(* CODESYS project Kontrolki2.project

Project tree, tasks and I/O mapping:
  Device : CODESYS Control Win V3, 3S - Smart Software Solutions GmbH, order no. 305021, version 3.5.8.10
    application Application
      libraries: Standard, * (System)
      task MainTask (cyclic, interval t#20ms, priority 1) calls PLC_PRG
      task VISU_TASK (cyclic, interval 100 ms, priority 31) calls VisuElems.Visu_Prg
      program PLC_PRG [LD]
      visualisation Visualization
  libraries: VisuSymbols, 3.5.8.0 (System)
  text list GlobalTextList
*)

// Device/Application/PLC_PRG
PROGRAM PLC_PRG
VAR
	SET: BOOL;
	RESET: BOOL;
	//KONTROLKA 1 - CZERWONY
	K1: BOOL;
	//KONTROLKA 2 - ZIELONY
	K2: BOOL;
	//KONTROLKA 3 - NIEBIESKI
	K3: BOOL;
	//KONTROLKA 4 - ŻÓŁTY
	K4: BOOL;
	HOLD: BOOL;
	//SPRAWDZENIE CZY SIĘ ŚWIECI K1
	C1: BOOL;
	//SPRAWDZENIE CZY SIĘ ŚWIECI K2
	C2: BOOL;
	//SPRAWDZENIE CZY SIĘ ŚWIECI K3
	C3: BOOL;
	//SPRAWDZENIE CZY SIĘ ŚWIECI K4
	C4: BOOL;
	TON_K1: TON;
	TON_K2: TON;
	TON_K3: TON;
	CZAS: TIME;
	//SPRAWDZENIE CZY NACIŚNIĘTO RESET
	CHECK: BOOL;
END_VAR
VAR // added by the converter: edge detectors and wires of the graphical bodies
    _w1, _w2 : BOOL;
END_VAR

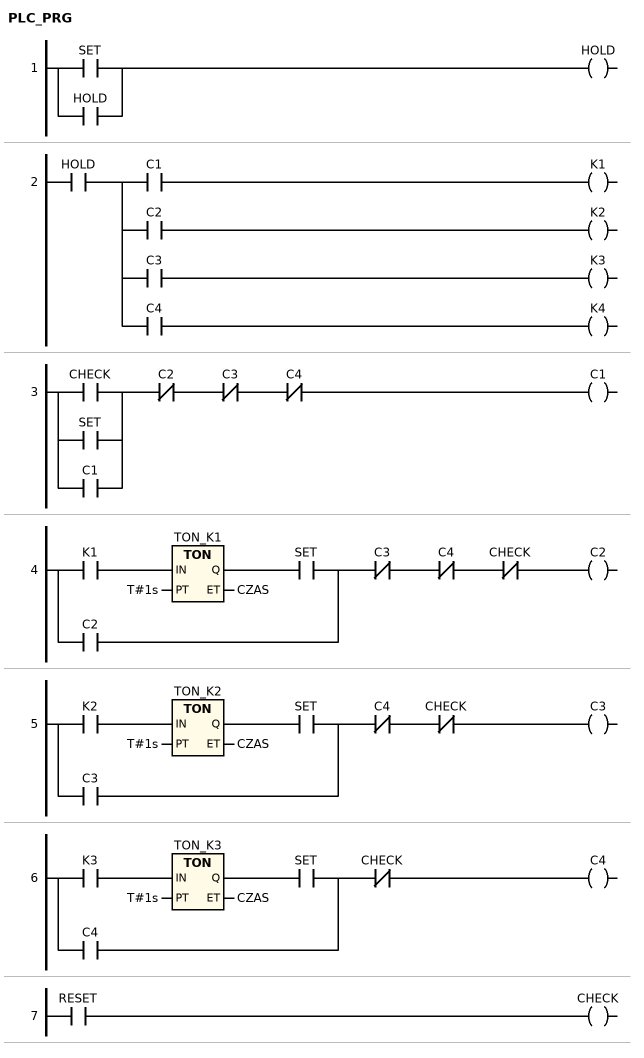
// NETWORK 1
HOLD := SET OR HOLD;

// NETWORK 2
K1 := HOLD AND C1;
K2 := HOLD AND C2;
K3 := HOLD AND C3;
K4 := HOLD AND C4;

// NETWORK 3
C1 := (CHECK OR SET OR C1) AND NOT C2 AND NOT C3 AND NOT C4;

// NETWORK 4
TON_K1(IN := K1, PT := T#1s, ET => CZAS); // TON
C2 := (TON_K1.Q AND SET OR C2) AND NOT C3 AND NOT C4 AND NOT CHECK;

// NETWORK 5
_w1 := C3;
IF NOT _w1 THEN
    TON_K2(IN := K2, PT := T#1s, ET => CZAS); // TON
    _w1 := TON_K2.Q AND SET;
END_IF
C3 := _w1 AND NOT C4 AND NOT CHECK;

// NETWORK 6
_w2 := C4;
IF NOT _w2 THEN
    TON_K3(IN := K3, PT := T#1s, ET => CZAS); // TON
    _w2 := TON_K3.Q AND SET;
END_IF
C4 := _w2 AND NOT CHECK;

// NETWORK 7
CHECK := RESET;

END_PROGRAM

// Device/Application/Visualization
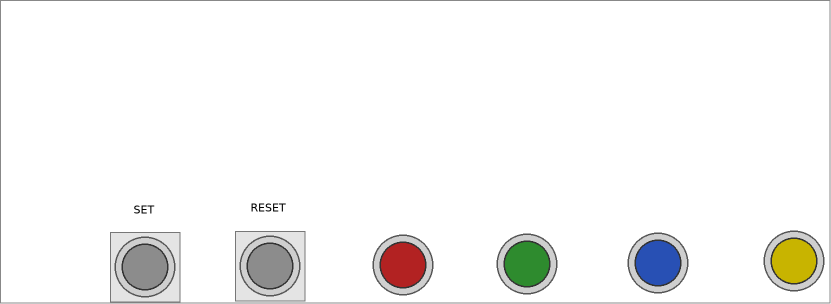
VISUALIZATION Visualization  // 831x304
    PushSwitch (110,232 70x70), variable: PLC_PRG.SET, behaviour: TAP, style: Switch-PushSwitch-Gray
    PushSwitch (235,231 70x70), variable: PLC_PRG.RESET, behaviour: TAP, style: Switch-PushSwitch-Gray
    Lamp1 (368,230 70x70), variable: PLC_PRG.K1, style: Lamp-Lamp1-Red
    Lamp1 (492,229 70x70), variable: PLC_PRG.K2, style: Lamp-Lamp1-Green
    Lamp1 (623,228 70x70), variable: PLC_PRG.K3, style: Lamp-Lamp1-Blue
    Lamp1 (759,226 70x70), variable: PLC_PRG.K4, style: Lamp-Lamp1-Yellow
    Label (69,195 150x30), "SET"
    Label (193,193 150x30), "RESET"
END_VISUALIZATION
